(* CODESYS project 车床桁架_RECOVERED_2024-04-08T08-30-31.project
   CompiledLibraryCompatibilityVersion: LeadSysStudio V3.5 SP15 Patch 4
   Title: 车床桁架

Project tree, tasks and I/O mapping:
  Device : SC5-C0A4, Leadshine Technology Co., Ltd., order no. 504001, version 3.5.15.40
    application Application
      libraries: Standard, * (System)
      task MainTask (cyclic, interval t#20ms, priority 1) calls PLC_PRG
      task EtherCAT_Master_Leadshine_A (cyclic, interval 4000 µs, priority 0) calls EtherCAT_Master_Leadshine_A.EtherCAT_Task
      FunctionBlock/
        function block FB102_ClockPuls [LD]
        program Public_Prog [LD]: SystemVar
        function block FB_CylinderDouble [ST]
        function block FB_CylinderSingle [ST]
      global variables HMI_Var
      global variables I_List
      data type CYLINDER_REF
      global variables System
      global variables Publics
      program PLC_PRG [LD]
      global variables O_Lisk
    Device Diagnose
    Network Configuration
      LocalBus Config
    Resource Usage
    LocalBus_Master_Module : LocalBusR1 Master, Leadshine Technology Co., Ltd., version 3.5.15.40
      SC0032N1 : SC0032N1, Leadshine Technology Co., Ltd., version 3.5.15.40
          settings: 位置号 = 1
          unmapped channels: OUTPUT_0, OUTPUT_1, OUTPUT_2, OUTPUT_3
      SC3200 : SC3200, Leadshine Technology Co., Ltd., version 3.5.15.40
          settings: 位置号 = 0
          unmapped channels: INPUT_0, INPUT_1, INPUT_2, INPUT_3
    SoftMotion General Axis Pool
    EtherCAT_Master_Leadshine_A : EtherCAT Master SoftMotion, 3S - Smart Software Solutions GmbH, version 3.5.16.30
        settings: NetworkName = 'ecat'; SelectNetworkByName = TRUE
      L6N_2 : L6N(COE), Leadshine Technology Co.,Ltd., order no. L6N, version Revision=16#00000001
          settings: DC sync0 cycletime = 4000; DC sync1 cycletime = 4000; Number of SDO = 6; Homing method.Index = 16#6098; Homing method.Subindex = 16#00; Homing method.Value = 19; Homing method.Size = 8; Homing method.AbortIfError = FALSE; Homing method.JumpToLine = FALSE; Homing method.Line = 0; Homing method.CompleteAccess = FALSE; Homing velocity (fast).Index = 16#6099; Homing velocity (fast).Subindex = 16#01; Homing velocity (fast).Value = 6103261; Homing velocity (fast).Size = 32; Homing velocity (fast).AbortIfError = FALSE; Homing velocity (fast).JumpToLine = FALSE; Homing velocity (fast).Line = 0; Homing velocity (fast).CompleteAccess = FALSE; Homing velocity (slow).Index = 16#6099; Homing velocity (slow).Subindex = 16#02; Homing velocity (slow).Value = 1220652; Homing velocity (slow).Size = 32; Homing velocity (slow).AbortIfError = FALSE; Homing velocity (slow).JumpToLine = FALSE; Homing velocity (slow).Line = 0; Homing velocity (slow).CompleteAccess = FALSE; Homing acceleration.Index = 16#609A; Homing acceleration.Subindex = 16#00; Homing acceleration.Value = 61032615; Homing acceleration.Size = 32; Homing acceleration.AbortIfError = FALSE; Homing acceleration.JumpToLine = FALSE; Homing acceleration.Line = 0; Homing acceleration.CompleteAccess = FALSE; Homing offset.Index = 16#607C; Homing offset.Subindex = 16#00; Homing offset.Value = 0; Homing offset.Size = 32; Homing offset.AbortIfError = FALSE;
            Homing offset.JumpToLine = FALSE; Homing offset.Line = 0; Homing offset.CompleteAccess = FALSE
          unmapped channels: Control word, Profile target position, Touch Probe Function, Last error code, Status word, Modes of operation display, Position loop error, Actual motor torque, Actual motor position, Touch Probe Status, Touch probe pos1 pos value, Digital inputs
        Axis_2 : Axis, 3S - Smart Software Solutions GmbH, order no. 0, version 4.6.1.0
            settings: wDriveID = 2; dwRatioTechUnitsDenom = 610326149; iRatioTechUnitsNum = 1000; fSWMaxVelocity = 1000; fSWMaxAcceleration = 10000; fSWMaxDeceleration = 10000; fSWMaxJerk = 100000; 一圈脉冲数 = 8388608; 工作台一圈的位移 = 109.955741; 电子齿轮比分子 = 8; 电子齿轮比分母 = 1; ScalingIncs = 8388608; ScalingMotorTurns2 = 8; AdrOffset_8010 = 28; BitOffset_8010 = 0; BitLength_8010 = 16; Address_8010 = '%QW14'; Type_8010 = 'UINT'; AddressPointer_8010 = ADR(%QW14); AdrOffset_8020 = 32; BitOffset_8020 = 0; BitLength_8020 = 32; Address_8020 = '%QD8'; Type_8020 = 'DINT'; AddressPointer_8020 = ADR(%QD8); AdrOffset_8030 = 4294967295; BitOffset_8030 = 0; BitLength_8030 = 32; Address_8030 = ''; Type_8030 = 'DINT'; AddressPointer_8030 = 0; AdrOffset_8040 = 4294967295; BitOffset_8040 = 0; BitLength_8040 = 16; Address_8040 = ''; Type_8040 = 'INT'; AddressPointer_8040 = 0; AdrOffset_8050 = 4294967295; BitOffset_8050 = 0; BitLength_8050 = 8;
              Address_8050 = ''; Type_8050 = 'SINT'; AddressPointer_8050 = 0; AdrOffset_8060 = 36; BitOffset_8060 = 0; BitLength_8060 = 16; Address_8060 = '%QW18'; Type_8060 = 'UINT'; AddressPointer_8060 = ADR(%QW18); AdrOffset_8070 = 4294967295; BitOffset_8070 = 0; BitLength_8070 = 0; Address_8070 = ''; Type_8070 = ''; AddressPointer_8070 = 0; AdrOffset_8080 = 4294967295; BitOffset_8080 = 0; BitLength_8080 = 16; Address_8080 = ''; Type_8080 = 'INT'; AddressPointer_8080 = 0; AdrOffset_8090 = 4294967295; BitOffset_8090 = 0; BitLength_8090 = 0; Address_8090 = ''; Type_8090 = ''; AddressPointer_8090 = 0; AdrOffset_8510 = 70; BitOffset_8510 = 0; BitLength_8510 = 16; Address_8510 = '%IW35'; Type_8510 = 'UINT'; AddressPointer_8510 = ADR(%IW35); AdrOffset_8520 = 84; BitOffset_8520 = 0; BitLength_8520 = 32; Address_8520 = '%ID21'; Type_8520 = 'DINT'; AddressPointer_8520 = ADR(%ID21); AdrOffset_8530 = 4294967295;
              BitOffset_8530 = 0; BitLength_8530 = 0; Address_8530 = ''; Type_8530 = ''; AddressPointer_8530 = 0; AdrOffset_8540 = 80; BitOffset_8540 = 0; BitLength_8540 = 16; Address_8540 = '%IW40'; Type_8540 = 'INT'; AddressPointer_8540 = ADR(%IW40); AdrOffset_8550 = 72; BitOffset_8550 = 0; BitLength_8550 = 8; Address_8550 = '%IB72'; Type_8550 = 'SINT'; AddressPointer_8550 = ADR(%IB72); AdrOffset_8560 = 96; BitOffset_8560 = 0; BitLength_8560 = 32; Address_8560 = '%ID24'; Type_8560 = 'UDINT'; AddressPointer_8560 = ADR(%ID24); AdrOffset_8570 = 88; BitOffset_8570 = 0; BitLength_8570 = 16; Address_8570 = '%IW44'; Type_8570 = 'UINT'; AddressPointer_8570 = ADR(%IW44); AdrOffset_8580 = 92; BitOffset_8580 = 0; BitLength_8580 = 32; Address_8580 = '%ID23'; Type_8580 = 'DINT'; AddressPointer_8580 = ADR(%ID23); AdrOffset_8590 = 4294967295; BitOffset_8590 = 0; BitLength_8590 = 0; Address_8590 = ''; Type_8590 = '';
              AddressPointer_8590 = 0; AdrOffset_8600 = 4294967295; BitOffset_8600 = 0; BitLength_8600 = 0; Address_8600 = ''; Type_8600 = ''; AddressPointer_8600 = 0; AdrOffset_8600 = 4294967295; BitOffset_8600 = 0; BitLength_8600 = 0; Address_8610 = ''; Type_8610 = ''; AddressPointer_8610 = 0; AdrOffset_8620 = 76; BitOffset_8620 = 0; BitLength_8620 = 32; Address_8620 = '%ID19'; Type_8620 = 'DINT'; AddressPointer_8620 = ADR(%ID19)
      L6N_3 : L6N(COE), Leadshine Technology Co.,Ltd., order no. L6N, version Revision=16#00000001
          settings: DC sync0 cycletime = 4000; DC sync1 cycletime = 4000; Number of SDO = 6; Homing method.Index = 16#6098; Homing method.Subindex = 16#00; Homing method.Value = 19; Homing method.Size = 8; Homing method.AbortIfError = FALSE; Homing method.JumpToLine = FALSE; Homing method.Line = 0; Homing method.CompleteAccess = FALSE; Homing velocity (fast).Index = 16#6099; Homing velocity (fast).Subindex = 16#01; Homing velocity (fast).Value = 26701769; Homing velocity (fast).Size = 32; Homing velocity (fast).AbortIfError = FALSE; Homing velocity (fast).JumpToLine = FALSE; Homing velocity (fast).Line = 0; Homing velocity (fast).CompleteAccess = FALSE; Homing velocity (slow).Index = 16#6099; Homing velocity (slow).Subindex = 16#02; Homing velocity (slow).Value = 5340354; Homing velocity (slow).Size = 32; Homing velocity (slow).AbortIfError = FALSE; Homing velocity (slow).JumpToLine = FALSE; Homing velocity (slow).Line = 0; Homing velocity (slow).CompleteAccess = FALSE; Homing acceleration.Index = 16#609A; Homing acceleration.Subindex = 16#00; Homing acceleration.Value = 267017690; Homing acceleration.Size = 32; Homing acceleration.AbortIfError = FALSE; Homing acceleration.JumpToLine = FALSE; Homing acceleration.Line = 0; Homing acceleration.CompleteAccess = FALSE; Homing offset.Index = 16#607C; Homing offset.Subindex = 16#00; Homing offset.Value = 0; Homing offset.Size = 32; Homing offset.AbortIfError = FALSE;
            Homing offset.JumpToLine = FALSE; Homing offset.Line = 0; Homing offset.CompleteAccess = FALSE
          unmapped channels: Control word, Profile target position, Touch Probe Function, Last error code, Status word, Modes of operation display, Position loop error, Actual motor torque, Actual motor position, Touch Probe Status, Touch probe pos1 pos value, Digital inputs
        Axis_3 : Axis, 3S - Smart Software Solutions GmbH, order no. 0, version 4.6.1.0
            settings: wDriveID = 3; dwRatioTechUnitsDenom = 26701769; iRatioTechUnitsNum = 10; fSWMaxVelocity = 1000; fSWMaxAcceleration = 10000; fSWMaxDeceleration = 10000; fSWMaxJerk = 100000; 一圈脉冲数 = 8388608; 工作台一圈的位移 = 109.955741; 电子齿轮比分子 = 35; 电子齿轮比分母 = 1; ScalingIncs = 8388608; ScalingMotorTurns2 = 35; AdrOffset_8010 = 40; BitOffset_8010 = 0; BitLength_8010 = 16; Address_8010 = '%QW20'; Type_8010 = 'UINT'; AddressPointer_8010 = ADR(%QW20); AdrOffset_8020 = 44; BitOffset_8020 = 0; BitLength_8020 = 32; Address_8020 = '%QD11'; Type_8020 = 'DINT'; AddressPointer_8020 = ADR(%QD11); AdrOffset_8030 = 4294967295; BitOffset_8030 = 0; BitLength_8030 = 32; Address_8030 = ''; Type_8030 = 'DINT'; AddressPointer_8030 = 0; AdrOffset_8040 = 4294967295; BitOffset_8040 = 0; BitLength_8040 = 16; Address_8040 = ''; Type_8040 = 'INT'; AddressPointer_8040 = 0; AdrOffset_8050 = 4294967295; BitOffset_8050 = 0; BitLength_8050 = 8;
              Address_8050 = ''; Type_8050 = 'SINT'; AddressPointer_8050 = 0; AdrOffset_8060 = 48; BitOffset_8060 = 0; BitLength_8060 = 16; Address_8060 = '%QW24'; Type_8060 = 'UINT'; AddressPointer_8060 = ADR(%QW24); AdrOffset_8070 = 4294967295; BitOffset_8070 = 0; BitLength_8070 = 0; Address_8070 = ''; Type_8070 = ''; AddressPointer_8070 = 0; AdrOffset_8080 = 4294967295; BitOffset_8080 = 0; BitLength_8080 = 16; Address_8080 = ''; Type_8080 = 'INT'; AddressPointer_8080 = 0; AdrOffset_8090 = 4294967295; BitOffset_8090 = 0; BitLength_8090 = 0; Address_8090 = ''; Type_8090 = ''; AddressPointer_8090 = 0; AdrOffset_8510 = 102; BitOffset_8510 = 0; BitLength_8510 = 16; Address_8510 = '%IW51'; Type_8510 = 'UINT'; AddressPointer_8510 = ADR(%IW51); AdrOffset_8520 = 116; BitOffset_8520 = 0; BitLength_8520 = 32; Address_8520 = '%ID29'; Type_8520 = 'DINT'; AddressPointer_8520 = ADR(%ID29); AdrOffset_8530 = 4294967295;
              BitOffset_8530 = 0; BitLength_8530 = 0; Address_8530 = ''; Type_8530 = ''; AddressPointer_8530 = 0; AdrOffset_8540 = 112; BitOffset_8540 = 0; BitLength_8540 = 16; Address_8540 = '%IW56'; Type_8540 = 'INT'; AddressPointer_8540 = ADR(%IW56); AdrOffset_8550 = 104; BitOffset_8550 = 0; BitLength_8550 = 8; Address_8550 = '%IB104'; Type_8550 = 'SINT'; AddressPointer_8550 = ADR(%IB104); AdrOffset_8560 = 128; BitOffset_8560 = 0; BitLength_8560 = 32; Address_8560 = '%ID32'; Type_8560 = 'UDINT'; AddressPointer_8560 = ADR(%ID32); AdrOffset_8570 = 120; BitOffset_8570 = 0; BitLength_8570 = 16; Address_8570 = '%IW60'; Type_8570 = 'UINT'; AddressPointer_8570 = ADR(%IW60); AdrOffset_8580 = 124; BitOffset_8580 = 0; BitLength_8580 = 32; Address_8580 = '%ID31'; Type_8580 = 'DINT'; AddressPointer_8580 = ADR(%ID31); AdrOffset_8590 = 4294967295; BitOffset_8590 = 0; BitLength_8590 = 0; Address_8590 = ''; Type_8590 = '';
              AddressPointer_8590 = 0; AdrOffset_8600 = 4294967295; BitOffset_8600 = 0; BitLength_8600 = 0; Address_8600 = ''; Type_8600 = ''; AddressPointer_8600 = 0; AdrOffset_8600 = 4294967295; BitOffset_8600 = 0; BitLength_8600 = 0; Address_8610 = ''; Type_8610 = ''; AddressPointer_8610 = 0; AdrOffset_8620 = 108; BitOffset_8620 = 0; BitLength_8620 = 32; Address_8620 = '%ID27'; Type_8620 = 'DINT'; AddressPointer_8620 = ADR(%ID27)
      L6N_1 : L6N(COE), Leadshine Technology Co.,Ltd., order no. L6N, version Revision=16#00000001
          settings: DC sync0 cycletime = 4000; DC sync1 cycletime = 4000; Number of SDO = 6; Homing method.Index = 16#6098; Homing method.Subindex = 16#00; Homing method.Value = 19; Homing method.Size = 8; Homing method.AbortIfError = FALSE; Homing method.JumpToLine = FALSE; Homing method.Line = 0; Homing method.CompleteAccess = FALSE; Homing velocity (fast).Index = 16#6099; Homing velocity (fast).Subindex = 16#01; Homing velocity (fast).Value = 16777216; Homing velocity (fast).Size = 32; Homing velocity (fast).AbortIfError = FALSE; Homing velocity (fast).JumpToLine = FALSE; Homing velocity (fast).Line = 0; Homing velocity (fast).CompleteAccess = FALSE; Homing velocity (slow).Index = 16#6099; Homing velocity (slow).Subindex = 16#02; Homing velocity (slow).Value = 3355443; Homing velocity (slow).Size = 32; Homing velocity (slow).AbortIfError = FALSE; Homing velocity (slow).JumpToLine = FALSE; Homing velocity (slow).Line = 0; Homing velocity (slow).CompleteAccess = FALSE; Homing acceleration.Index = 16#609A; Homing acceleration.Subindex = 16#00; Homing acceleration.Value = 167772160; Homing acceleration.Size = 32; Homing acceleration.AbortIfError = FALSE; Homing acceleration.JumpToLine = FALSE; Homing acceleration.Line = 0; Homing acceleration.CompleteAccess = FALSE; Homing offset.Index = 16#607C; Homing offset.Subindex = 16#00; Homing offset.Value = 0; Homing offset.Size = 32; Homing offset.AbortIfError = FALSE;
            Homing offset.JumpToLine = FALSE; Homing offset.Line = 0; Homing offset.CompleteAccess = FALSE
          unmapped channels: Control word, Profile target position, Touch Probe Function, Last error code, Status word, Modes of operation display, Position loop error, Actual motor torque, Actual motor position, Touch Probe Status, Touch probe pos1 pos value, Digital inputs
        Axis_1 : Axis, 3S - Smart Software Solutions GmbH, order no. 0, version 4.6.1.0
            settings: dwRatioTechUnitsDenom = 8388608; iRatioTechUnitsNum = 5; fSWMaxVelocity = 1000; fSWMaxAcceleration = 10000; fSWMaxDeceleration = 10000; fSWMaxJerk = 100000; 一圈脉冲数 = 8388608; 工作台一圈的位移 = 5; 电子齿轮比分子 = 1; 电子齿轮比分母 = 1; ScalingIncs = 8388608; AdrOffset_8010 = 16; BitOffset_8010 = 0; BitLength_8010 = 16; Address_8010 = '%QW8'; Type_8010 = 'UINT'; AddressPointer_8010 = ADR(%QW8); AdrOffset_8020 = 20; BitOffset_8020 = 0; BitLength_8020 = 32; Address_8020 = '%QD5'; Type_8020 = 'DINT'; AddressPointer_8020 = ADR(%QD5); AdrOffset_8030 = 4294967295; BitOffset_8030 = 0; BitLength_8030 = 32; Address_8030 = ''; Type_8030 = 'DINT'; AddressPointer_8030 = 0; AdrOffset_8040 = 4294967295; BitOffset_8040 = 0; BitLength_8040 = 16; Address_8040 = ''; Type_8040 = 'INT'; AddressPointer_8040 = 0; AdrOffset_8050 = 4294967295; BitOffset_8050 = 0; BitLength_8050 = 8; Address_8050 = ''; Type_8050 = 'SINT';
              AddressPointer_8050 = 0; AdrOffset_8060 = 24; BitOffset_8060 = 0; BitLength_8060 = 16; Address_8060 = '%QW12'; Type_8060 = 'UINT'; AddressPointer_8060 = ADR(%QW12); AdrOffset_8070 = 4294967295; BitOffset_8070 = 0; BitLength_8070 = 0; Address_8070 = ''; Type_8070 = ''; AddressPointer_8070 = 0; AdrOffset_8080 = 4294967295; BitOffset_8080 = 0; BitLength_8080 = 16; Address_8080 = ''; Type_8080 = 'INT'; AddressPointer_8080 = 0; AdrOffset_8090 = 4294967295; BitOffset_8090 = 0; BitLength_8090 = 0; Address_8090 = ''; Type_8090 = ''; AddressPointer_8090 = 0; AdrOffset_8510 = 38; BitOffset_8510 = 0; BitLength_8510 = 16; Address_8510 = '%IW19'; Type_8510 = 'UINT'; AddressPointer_8510 = ADR(%IW19); AdrOffset_8520 = 52; BitOffset_8520 = 0; BitLength_8520 = 32; Address_8520 = '%ID13'; Type_8520 = 'DINT'; AddressPointer_8520 = ADR(%ID13); AdrOffset_8530 = 4294967295; BitOffset_8530 = 0; BitLength_8530 = 0;
              Address_8530 = ''; Type_8530 = ''; AddressPointer_8530 = 0; AdrOffset_8540 = 48; BitOffset_8540 = 0; BitLength_8540 = 16; Address_8540 = '%IW24'; Type_8540 = 'INT'; AddressPointer_8540 = ADR(%IW24); AdrOffset_8550 = 40; BitOffset_8550 = 0; BitLength_8550 = 8; Address_8550 = '%IB40'; Type_8550 = 'SINT'; AddressPointer_8550 = ADR(%IB40); AdrOffset_8560 = 64; BitOffset_8560 = 0; BitLength_8560 = 32; Address_8560 = '%ID16'; Type_8560 = 'UDINT'; AddressPointer_8560 = ADR(%ID16); AdrOffset_8570 = 56; BitOffset_8570 = 0; BitLength_8570 = 16; Address_8570 = '%IW28'; Type_8570 = 'UINT'; AddressPointer_8570 = ADR(%IW28); AdrOffset_8580 = 60; BitOffset_8580 = 0; BitLength_8580 = 32; Address_8580 = '%ID15'; Type_8580 = 'DINT'; AddressPointer_8580 = ADR(%ID15); AdrOffset_8590 = 4294967295; BitOffset_8590 = 0; BitLength_8590 = 0; Address_8590 = ''; Type_8590 = ''; AddressPointer_8590 = 0; AdrOffset_8600 = 4294967295;
              BitOffset_8600 = 0; BitLength_8600 = 0; Address_8600 = ''; Type_8600 = ''; AddressPointer_8600 = 0; AdrOffset_8600 = 4294967295; BitOffset_8600 = 0; BitLength_8600 = 0; Address_8610 = ''; Type_8610 = ''; AddressPointer_8610 = 0; AdrOffset_8620 = 44; BitOffset_8620 = 0; BitLength_8620 = 32; Address_8620 = '%ID11'; Type_8620 = 'DINT'; AddressPointer_8620 = ADR(%ID11)
      L6N : L6N(COE), Leadshine Technology Co.,Ltd., order no. L6N, version Revision=16#00000001
          settings: DC sync0 cycletime = 4000; DC enable = 1; DC sync0 enable = 1; DC sync0 shift time = 0; DC sync1 cycletime = 4000; DC sync1 enable = 0; DC sync1 factor = 'x 1'; DC sync1 shift time = 0; Number of SDO = 6; Homing method.Index = 16#6098; Homing method.Subindex = 16#00; Homing method.Value = 30; Homing method.Size = 8; Homing method.AbortIfError = FALSE; Homing method.JumpToLine = FALSE; Homing method.Line = 0; Homing method.CompleteAccess = FALSE; Homing velocity (fast).Index = 16#6099; Homing velocity (fast).Subindex = 16#01; Homing velocity (fast).Value = 20971520; Homing velocity (fast).Size = 32; Homing velocity (fast).AbortIfError = FALSE; Homing velocity (fast).JumpToLine = FALSE; Homing velocity (fast).Line = 0; Homing velocity (fast).CompleteAccess = FALSE; Homing velocity (slow).Index = 16#6099; Homing velocity (slow).Subindex = 16#02; Homing velocity (slow).Value = 4194304; Homing velocity (slow).Size = 32; Homing velocity (slow).AbortIfError = FALSE; Homing velocity (slow).JumpToLine = FALSE; Homing velocity (slow).Line = 0; Homing velocity (slow).CompleteAccess = FALSE; Homing acceleration.Index = 16#609A; Homing acceleration.Subindex = 16#00; Homing acceleration.Value = 209715200; Homing acceleration.Size = 32; Homing acceleration.AbortIfError = FALSE; Homing acceleration.JumpToLine = FALSE; Homing acceleration.Line = 0;
            Homing acceleration.CompleteAccess = FALSE; Homing offset.Index = 16#607C; Homing offset.Subindex = 16#00; Homing offset.Value = 0; Homing offset.Size = 32; Homing offset.AbortIfError = FALSE; Homing offset.JumpToLine = FALSE; Homing offset.Line = 0; Homing offset.CompleteAccess = FALSE
          unmapped channels: Control word, Profile target position, Touch Probe Function, Last error code, Status word, Modes of operation display, Position loop error, Actual motor torque, Actual motor position, Touch Probe Status, Touch probe pos1 pos value, Digital inputs
        Axis : Axis, 3S - Smart Software Solutions GmbH, order no. 0, version 4.6.1.0
            settings: wDriveID = 0; dwRatioTechUnitsDenom = 2097152; fSWMaxVelocity = 1000; fSWMaxAcceleration = 10000; fSWMaxDeceleration = 10000; fSWMaxJerk = 100000; 一圈脉冲数 = 8388608; 工作台一圈的位移 = 4; 电子齿轮比分子 = 1; 电子齿轮比分母 = 1; ScalingIncs = 8388608; AdrOffset_8010 = 4; BitOffset_8010 = 0; BitLength_8010 = 16; Address_8010 = '%QW2'; Type_8010 = 'UINT'; AddressPointer_8010 = ADR(%QW2); AdrOffset_8020 = 8; BitOffset_8020 = 0; BitLength_8020 = 32; Address_8020 = '%QD2'; Type_8020 = 'DINT'; AddressPointer_8020 = ADR(%QD2); AdrOffset_8030 = 4294967295; BitOffset_8030 = 0; BitLength_8030 = 32; Address_8030 = ''; Type_8030 = 'DINT'; AddressPointer_8030 = 0; AdrOffset_8040 = 4294967295; BitOffset_8040 = 0; BitLength_8040 = 16; Address_8040 = ''; Type_8040 = 'INT'; AddressPointer_8040 = 0; AdrOffset_8050 = 4294967295; BitOffset_8050 = 0; BitLength_8050 = 8; Address_8050 = ''; Type_8050 = 'SINT';
              AddressPointer_8050 = 0; AdrOffset_8060 = 12; BitOffset_8060 = 0; BitLength_8060 = 16; Address_8060 = '%QW6'; Type_8060 = 'UINT'; AddressPointer_8060 = ADR(%QW6); AdrOffset_8070 = 4294967295; BitOffset_8070 = 0; BitLength_8070 = 0; Address_8070 = ''; Type_8070 = ''; AddressPointer_8070 = 0; AdrOffset_8080 = 4294967295; BitOffset_8080 = 0; BitLength_8080 = 16; Address_8080 = ''; Type_8080 = 'INT'; AddressPointer_8080 = 0; AdrOffset_8090 = 4294967295; BitOffset_8090 = 0; BitLength_8090 = 0; Address_8090 = ''; Type_8090 = ''; AddressPointer_8090 = 0; AdrOffset_8510 = 6; BitOffset_8510 = 0; BitLength_8510 = 16; Address_8510 = '%IW3'; Type_8510 = 'UINT'; AddressPointer_8510 = ADR(%IW3); AdrOffset_8520 = 20; BitOffset_8520 = 0; BitLength_8520 = 32; Address_8520 = '%ID5'; Type_8520 = 'DINT'; AddressPointer_8520 = ADR(%ID5); AdrOffset_8530 = 4294967295; BitOffset_8530 = 0; BitLength_8530 = 0;
              Address_8530 = ''; Type_8530 = ''; AddressPointer_8530 = 0; AdrOffset_8540 = 16; BitOffset_8540 = 0; BitLength_8540 = 16; Address_8540 = '%IW8'; Type_8540 = 'INT'; AddressPointer_8540 = ADR(%IW8); AdrOffset_8550 = 8; BitOffset_8550 = 0; BitLength_8550 = 8; Address_8550 = '%IB8'; Type_8550 = 'SINT'; AddressPointer_8550 = ADR(%IB8); AdrOffset_8560 = 32; BitOffset_8560 = 0; BitLength_8560 = 32; Address_8560 = '%ID8'; Type_8560 = 'UDINT'; AddressPointer_8560 = ADR(%ID8); AdrOffset_8570 = 24; BitOffset_8570 = 0; BitLength_8570 = 16; Address_8570 = '%IW12'; Type_8570 = 'UINT'; AddressPointer_8570 = ADR(%IW12); AdrOffset_8580 = 28; BitOffset_8580 = 0; BitLength_8580 = 32; Address_8580 = '%ID7'; Type_8580 = 'DINT'; AddressPointer_8580 = ADR(%ID7); AdrOffset_8590 = 4294967295; BitOffset_8590 = 0; BitLength_8590 = 0; Address_8590 = ''; Type_8590 = ''; AddressPointer_8590 = 0; AdrOffset_8600 = 4294967295;
              BitOffset_8600 = 0; BitLength_8600 = 0; Address_8600 = ''; Type_8600 = ''; AddressPointer_8600 = 0; AdrOffset_8600 = 4294967295; BitOffset_8600 = 0; BitLength_8600 = 0; Address_8610 = ''; Type_8610 = ''; AddressPointer_8610 = 0; AdrOffset_8620 = 12; BitOffset_8620 = 0; BitLength_8620 = 32; Address_8620 = '%ID3'; Type_8620 = 'DINT'; AddressPointer_8620 = ADR(%ID3)
*)

// Device/Application/CYLINDER_REF
TYPE CYLINDER_REF :
STRUCT
	///初始化时返回原位控制
	xInit: BOOL;
	///自动控制,变为TRUE时，执行到位控制，变为FALSE时执行原位控制
	xAutoCmd: BOOL;
	///到位标志,处于原位状态
	xIsBack: BOOL;
	///到位标志,处于到位状态	
	xIsFront: BOOL;
END_STRUCT
END_TYPE

// Device/Application/HMI_Var
{attribute 'qualified_only'}
VAR_GLOBAL
END_VAR

// Device/Application/I_List
{attribute 'qualified_only'}
VAR_GLOBAL
	// 上料传送带到位确认
	X0 AT %IX0.0: BOOL;
	// 紧急停止
	X1 AT %IX0.1: BOOL;
	// 推出气缸原位
	X2 AT %IX0.2: BOOL;
	// 推出气缸动作位
	X3 AT %IX0.3: BOOL;
	// 顶起气缸原位
	X4 AT %IX0.4: BOOL;
	// 顶起气缸动作位
	X5 AT %IX0.5: BOOL;
	// 上料气爪原位
	X6 AT %IX0.6: BOOL;
	// 上料气爪动作位
	X7 AT %IX0.7: BOOL;
	// 下料气爪原位
	X10 AT %IX1.0: BOOL;
	// 下料气爪动作位
	X11 AT %IX1.1: BOOL;
	// 翻转气缸原位
	X12 AT %IX1.2: BOOL;
	// 翻转气缸动作位
	X13 AT %IX1.3: BOOL;
	// 开门气缸原位
	X14 AT %IX1.4: BOOL;
	// 开门气缸动作位
	X15 AT %IX1.5: BOOL;
	// 启动按钮
	X16 AT %IX1.6: BOOL;
	// 停止按钮
	X17 AT %IX1.7: BOOL;
	// 复位按钮
	X20 AT %IX2.0: BOOL;
	// 手自动按钮ON为自动
	X21 AT %IX2.1: BOOL;
	// 下料确认
	X22 AT %IX2.2: BOOL;
	// 联机卡盘夹紧
	X23 AT %IX2.3: BOOL;
	// 联机启动
	X24 AT %IX2.4: BOOL;
	// 联机停止
	X25 AT %IX2.5: BOOL;
	// 联机故障
	X26 AT %IX2.6: BOOL;
	// 联机X轴零点
	X27 AT %IX2.7: BOOL;
	// 联机Z轴零点
	X30 AT %IX3.0: BOOL;
	X31 AT %IX3.1: BOOL;
	X32 AT %IX3.2: BOOL;
	X33 AT %IX3.3: BOOL;
	X34 AT %IX3.4: BOOL;
	X35 AT %IX3.5: BOOL;
	X36 AT %IX3.6: BOOL;
	X37 AT %IX3.7: BOOL;
END_VAR

// Device/Application/System
{attribute 'qualified_only'}
VAR_GLOBAL
	// 上电扫描一周期
FirstScan    :BOOL;
// 常ON
AlwaysTRUE   : BOOL;
// 常OFF
AlwaysFALSE  : BOOL;
// 0.1S周期脉冲
Clock_10Hz    :BOOL;
// 0.2S周期脉冲
Clock_5Hz    :BOOL;
// 0.5S周期脉冲
Clock_2Hz    :BOOL;
// 1S周期脉冲
Clock_1Hz    :BOOL;
// 2S周期脉冲
Clock_HalfHz :BOOL;
END_VAR

// Device/Application/Publics
{attribute 'qualified_only'}
VAR_GLOBAL
	// 调试使用常ON
CYGIA_ON   :BOOL;
// 调试使用常OFF
CYGIA_OFF  :BOOL;
END_VAR

// Device/Application/O_Lisk
{attribute 'qualified_only'}
VAR_GLOBAL
	// 皮带运转
	Y0 AT %QX0.0: BOOL;
	// 震动筛运动
	Y1 AT %QX0.1: BOOL;
	// 推出气缸原位
	Y2 AT %QX0.2: BOOL;
	// 紧急停止输出
	Y3 AT %QX0.3: BOOL;
	// 顶起气缸原位
	Y4 AT %QX0.4: BOOL;
	Y5 AT %QX0.5: BOOL;
	// 上料气爪原位
	Y6 AT %QX0.6: BOOL;
	Y7 AT %QX0.7: BOOL;
	// 下料气爪原位
	Y10 AT %QX1.0: BOOL;
	Y11 AT %QX1.0: BOOL;
	// 翻转气缸原位
	Y12 AT %QX1.0: BOOL;
	Y13 AT %QX1.0: BOOL;
	// 开门气缸原位
	Y14 AT %QX1.0: BOOL;
	Y15 AT %QX1.5: BOOL;
	// 启动按钮LED
	Y16 AT %QX1.6: BOOL;
	// 停止按钮LED
	Y17 AT %QX1.7: BOOL;
	// 复位按钮LED
	Y20 AT %QX2.0: BOOL;
	Y21 AT %QX2.1: BOOL;
	// 下料传送带
	Y22 AT %QX2.2: BOOL;
	// 三色灯红
	Y23 AT %QX2.3: BOOL;
	// 三色灯黄
	Y24 AT %QX2.4: BOOL;
	// 三色灯绿
	Y25 AT %QX2.5: BOOL;
	// 三色灯蜂鸣
	Y26 AT %QX2.6: BOOL;
	// 联机卡盘夹紧
	Y27 AT %QX2.7: BOOL;
	// 联机启动
	Y30 AT %QX3.0: BOOL;
	// 联机停止
	Y31 AT %QX3.1: BOOL;
	Y32 AT %QX3.2: BOOL;
	Y33 AT %QX3.3: BOOL;
	Y34 AT %QX3.4: BOOL;
	Y35 AT %QX3.5: BOOL;
	Y36 AT %QX3.6: BOOL;
	Y37 AT %QX3.7: BOOL;
END_VAR

// Device/Application/PLC_PRG
PROGRAM PLC_PRG
VAR
	SMC3_ReinitDrive_0: SMC3_ReinitDrive;
END_VAR

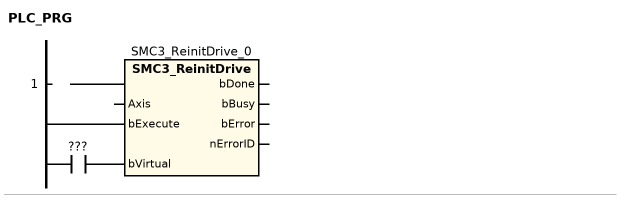
// NETWORK 1
SMC3_ReinitDrive_0(bExecute := TRUE); // SMC3_ReinitDrive

END_PROGRAM

// Device/Application/FunctionBlock/FB102_ClockPuls
FUNCTION_BLOCK FB102_ClockPuls
VAR_INPUT
	///脉冲ON时间
	iTimeON: TIME;
	///脉冲OFF时间
	iTimeOFF: TIME;
END_VAR
VAR_OUTPUT
	///时钟脉冲差速器
	oClockVar: BOOL;
END_VAR
VAR
	TON_Clock: TON;
	TOF_Clock: TOF;
END_VAR

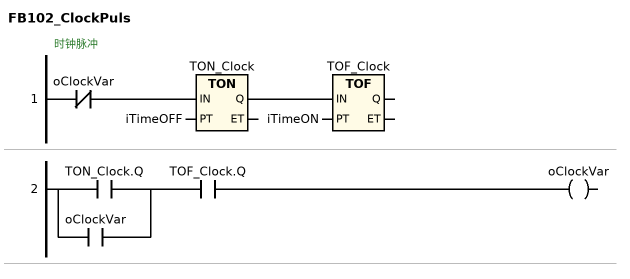
// NETWORK 1
// 时钟脉冲
TON_Clock(IN := NOT oClockVar, PT := iTimeOFF); // TON
TOF_Clock(IN := TON_Clock.Q, PT := iTimeON); // TOF

// NETWORK 2
oClockVar := (TON_Clock.Q OR oClockVar) AND TOF_Clock.Q;

END_FUNCTION_BLOCK

// Device/Application/FunctionBlock/Public_Prog
PROGRAM Public_Prog
VAR
	Clock_10Hz: FB102_ClockPuls;
	Clock_5Hz: FB102_ClockPuls;
	Clock_2Hz: FB102_ClockPuls;
	Clock_1Hz: FB102_ClockPuls;
	Clock_HalfHz: FB102_ClockPuls;
END_VAR
VAR // added by the converter: edge detectors and wires of the graphical bodies
    _rt1 : R_TRIG;
END_VAR

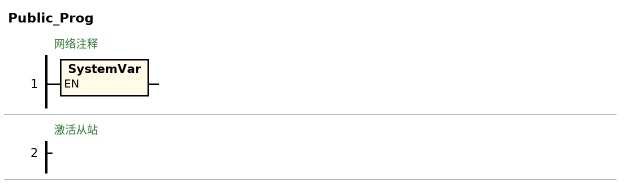
// NETWORK 1
// 网络注释
SystemVar();

// NETWORK 2
// 激活从站

ACTION SystemVar:
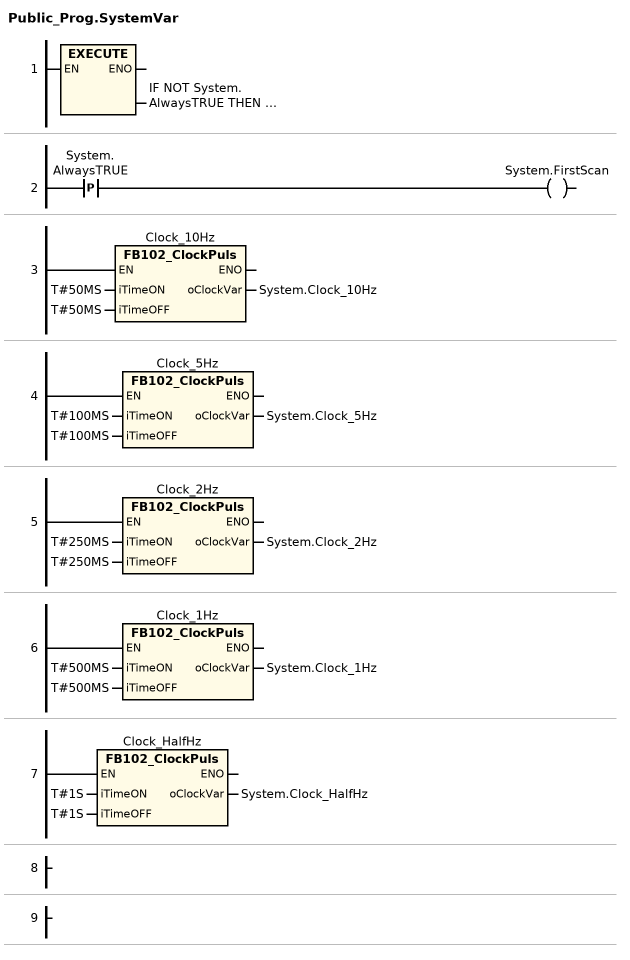
// NETWORK 1
IF NOT System.AlwaysTRUE THEN
	System.AlwaysTRUE := TRUE;
END_IF
IF  System.AlwaysFALSE THEN
	System.AlwaysFALSE := FALSE;
END_IF
IF NOT Publics.CYGIA_ON THEN
	Publics.CYGIA_ON := TRUE;
END_IF
IF  Publics.CYGIA_OFF THEN
	Publics.CYGIA_OFF := FALSE;
END_IF

// NETWORK 2
_rt1(CLK := System.AlwaysTRUE);
System.FirstScan := _rt1.Q;

// NETWORK 3
Clock_10Hz(iTimeON := T#50MS, iTimeOFF := T#50MS, oClockVar => System.Clock_10Hz); // FB102_ClockPuls

// NETWORK 4
Clock_5Hz(iTimeON := T#100MS, iTimeOFF := T#100MS, oClockVar => System.Clock_5Hz); // FB102_ClockPuls

// NETWORK 5
Clock_2Hz(iTimeON := T#250MS, iTimeOFF := T#250MS, oClockVar => System.Clock_2Hz); // FB102_ClockPuls

// NETWORK 6
Clock_1Hz(iTimeON := T#500MS, iTimeOFF := T#500MS, oClockVar => System.Clock_1Hz); // FB102_ClockPuls

// NETWORK 7
Clock_HalfHz(iTimeON := T#1S, iTimeOFF := T#1S, oClockVar => System.Clock_HalfHz); // FB102_ClockPuls

// NETWORK 8

// NETWORK 9
END_ACTION

END_PROGRAM

// Device/Application/FunctionBlock/FB_CylinderDouble
FUNCTION_BLOCK FB_CylinderDouble
VAR_IN_OUT
	///气缸控制、状态和报警
	stCylvar: CYLINDER_REF;
END_VAR
VAR_INPUT
	///安全条件
	xReady: BOOL;
	///报警复位
	xReset: BOOL;
	///手动控制,每on一次,则反转输出点状态
	xManuCmd: BOOL;
	///原位检测
	xBackSensor: BOOL;
	///到位检测
	xFrontSensor: BOOL;
	///手自动不一致报警无效
	xManuAlmDisable: BOOL;
	///原位检测无效
	xBackSensorDisable: BOOL;
	///到位检测无效	
	xFrontSensorDisable: BOOL;
	///原位延时	
	wBackDelay: WORD;
	///到位延时
	wFrontDelay: WORD;
END_VAR
VAR_OUTPUT
	///输出点,对应双控气缸原位电磁阀
	xOutputA: BOOL;
	///输出点,应双控气缸到位电磁阀
	xOutputB: BOOL;
	///未满足安全条件报警
	f_xNotRdyAlm: BOOL;
	///手自动不一致报警	
	f_xManuAlm: BOOL;
	///未在原位报警
	f_xBackAlm: BOOL;
	///未到位报警	
	f_xFrontAlm: BOOL;
	///气缸处于不受控制状态报警
	f_xUncontrolledAlm: BOOL;
END_VAR
VAR
	///获取自动控制的上升沿
	fbAutoRise: R_TRIG;
	///获取自动控制的下升沿
	fbAutoFall: F_TRIG;
	///获取手动控制的下升沿
	fbManuFall: F_TRIG;
	///获取复位信号的上升沿
	fbResetRise: R_TRIG;
	///原位状态延时,用于输出原位状态
	fbBackTon: TON;
	///到位状态延时,用于输出到位状态	
	fbFrontTon: TON;
	///获取原位状态下降沿
	fbBackFall: F_TRIG;
	///获取到位状态下降沿
	fbFrontFall: F_TRIG;
	///原位动作超时,用于输出未在原位位置报警
	fbBackWait: TON;
	///到位动作超时,用于输出未在原位位置报警
	fbFrontWait: TON;
END_VAR

   //初始化时返回原位
   IF  xReady AND stCylvar.xInit AND ( NOT xManuCmd ) THEN
	     xOutputA  := TRUE; 
         xOutputB  := FALSE;
		 f_xManuAlm  := FALSE;
		 stCylvar.xInit  := FALSE;	  	  	 	  
   END_IF	  
   
   //获取手动控制、自动控制的边沿信号
   fbManuFall(CLK:=xManuCmd , Q=> );
   fbAutoRise(CLK:=stCylvar.xAutoCmd , Q=> );
   fbAutoFall(CLK:=stCylvar.xAutoCmd , Q=> );
   
   //1,手动操作时，如果满足安全条件且未屏蔽手自动不一致报警时，则输出点A反转，输出点B取输出点A的反逻辑
   IF xReady AND (NOT xManuAlmDisable) AND fbManuFall.Q THEN
	   xOutputA  := NOT xOutputA; 
	   xOutputB  := NOT xOutputA;
	   
	//手动操作生效时，判断输出点状态与自动命令是否一致，不一致时,置位手动操作执行中报警；一致时复位该报警。
	//当因安全条件不满足导致自动命令未执行时，可通过手动操作控制其动作执行,此时手动操作并不引起手动操作执行中报警。
   	   IF (stCylvar.xAutoCmd AND (NOT xManuAlmDisable) ) XOR xOutputB THEN
   	   	    f_xManuAlm  :=TRUE;
   	   ELSE 
   	   	    f_xManuAlm  :=FALSE;
   	   END_IF
   END_IF
   //2,手动操作时，如果满足安全条件且屏蔽了手自动不一致报警时，则自动控制点反转、复位手自动不一致报警，  
    IF xReady AND  xManuAlmDisable AND fbManuFall.Q THEN
   	    stCylvar.xAutoCmd  := NOT stCylvar.xAutoCmd ;
		f_xManuAlm  :=FALSE;		  	 	
    END_IF
   
   //自动命令置位时，如满足安全条件，则输出点A复位、 输出点B置位。
   IF xReady AND fbAutoRise.Q THEN
   	    xOutputA  :=FALSE;
		xOutputB  :=TRUE;
		
   END_IF
   //自动命令复位时，如满足安全条件，则输出点A置位、 输出点B复位。
   IF xReady AND fbAutoFall.Q THEN
   	    xOutputA  :=TRUE;
		xOutputB  :=FALSE;		
   END_IF
   
   
   //到位状态输出
   fbFrontTon(IN:=( NOT xOutputA ) AND xOutputB AND ( xFrontSensor OR xFrontSensorDisable ) AND ( NOT xBackSensor ) , PT:= WORD_TO_TIME ( wFrontDelay *10 ), Q=> stCylvar.xIsFront, ET=> );
   
   //原位状态输出
   fbBackTon(IN:= xOutputA  AND ( NOT xOutputB) AND ( NOT xFrontSensor ) AND ( xBackSensor OR xBackSensorDisable ) , PT:= WORD_TO_TIME ( wBackDelay *10 ) , Q=> stCylvar.xIsBack, ET=> );
   
   
   //报警复位
   fbResetRise(CLK:= xReset, Q=> );
   IF fbResetRise.Q THEN
   	   f_xNotRdyAlm := FALSE;
	   f_xFrontAlm := FALSE;
	   f_xBackAlm := FALSE;
	   f_xUncontrolledAlm := FALSE;
   
   END_IF
   
   
   //未满足安全条件报警
   //当手动操作或自动命令状态发生改变时，如果不能满足安全条件，则输出未满足安全条件报警
   IF ( fbManuFall.Q OR fbAutoRise.Q OR fbAutoFall.Q ) AND ( NOT xReady ) THEN
   	   f_xNotRdyAlm := TRUE; 
   END_IF
   
   
   //未在原位报警
   //自动命令变OFF后(上电后气缸处于自由状态时不判断)，延时5秒，如果原位标志未变为ON、且未发生手动操作和安全条件报警，则输出未到原位报警
   fbBackWait(IN:= ( NOT stCylvar.xAutoCmd ) AND ( xOutputA OR xOutputB ) , PT:= T#5S , Q=> , ET=> );
   fbBackFall(CLK:= stCylvar.xIsBack , Q=> );
   IF (( fbBackWait.Q AND (NOT stCylvar.xIsBack )) OR (( NOT stCylvar.xAutoCmd ) AND fbBackFall.Q )) AND  ( NOT f_xManuAlm ) AND  ( NOT f_xNotRdyAlm ) THEN
   	    f_xBackAlm := TRUE;
   END_IF
   
   
   //未在到位报警
   //自动命令变ON后，延时5秒，如果到位标志未变为ON、且未发生手动操作和安全条件报警，则输出未到位报警
   fbFrontWait(IN:= stCylvar.xAutoCmd , PT:= T#5S , Q=> , ET=> );
   fbFrontFall(CLK:= stCylvar.xIsFront, Q=> );
   IF ( ( fbFrontWait.Q AND ( NOT stCylvar.xIsFront ) ) OR (stCylvar.xAutoCmd AND fbFrontFall.Q )) AND ( NOT f_xManuAlm ) AND ( NOT f_xNotRdyAlm ) THEN
   	    f_xFrontAlm := TRUE;   
   END_IF      
   
   
   //不受控状态报警
   IF NOT ( xOutputA OR xOutputB ) THEN
   	    f_xUncontrolledAlm := TRUE;
   END_IF

END_FUNCTION_BLOCK

// Device/Application/FunctionBlock/FB_CylinderSingle
FUNCTION_BLOCK FB_CylinderSingle
VAR_IN_OUT
	stCylVar: CYLINDER_REF;
END_VAR
VAR_INPUT
	///安全条件
	xReady: BOOL;
	///报警复位
	xReset: BOOL;
	///手动控制,每on一次,则反转输出点状态
	xManuCmd: BOOL;
	///原位检测
	xBackSensor: BOOL;
	///到位检测
	xFrontSensor: BOOL;
	///手自动不一致报警无效
	xManuAlmDisable: BOOL;
	///原位检测无效
	xBackSensorDisable: BOOL;
	///到位检测无效
	xFrontSensorDisable: BOOL;
	///原位延时
	wBackDelay: WORD;
	///到位延时
	wFrontDelay: WORD;
END_VAR
VAR_OUTPUT
	xOutput: BOOL;
	///未满足安全条件报警
	f_xNotRdyAlm: BOOL;
	///手自动不一致报警	
	f_xManuAlm: BOOL;
	///未在原位报警
	f_xBackAlm: BOOL;
	///未到位报警
	f_xFrontAlm: BOOL;
END_VAR
VAR
	///获取自动控制的上升沿
	fbAutoRise: R_TRIG;
	///获取自动控制的下升沿
	fbAutoFall: F_TRIG;
	///获取手动控制的下升沿
	fbManuFall: F_TRIG;
	///获取复位信号的上升沿
	fbResetRise: R_TRIG;
	///原位状态延时,用于输出原位状态
	fbBackTon: TON;
	///到位状态延时,用于输出到位状态
	fbFrontTon: TON;
	///获取原位状态下降沿	
	fbBackFall: F_TRIG;
	///获取到位状态下降沿
	fbFrontFall: F_TRIG;
	///原位动作超时,用于输出未在原位位置报警
	fbBackWait: TON;
	///到位动作超时,用于输出未在到位位置报警
	fbFrontWait: TON;
END_VAR

   //初始化时复位输出点
   IF xReady AND stCylVar.xInit AND ( NOT f_xNotRdyAlm	) THEN
	    xOutput := FALSE;
	    f_xManuAlm  := FALSE;
	    stCylVar.xInit  := FALSE;
 
   END_IF


   //获取手动控制、自动控制的边沿信号
   fbManuFall(CLK:=xManuCmd , Q=> );
   fbAutoRise(CLK:=stCylvar.xAutoCmd , Q=> );
   fbAutoFall(CLK:=stCylvar.xAutoCmd , Q=> );
      
    //1,手动操作时，如果满足安全条件且未屏蔽了手自动不一致报警时，则输出点反转，  
    IF xReady AND (NOT xManuAlmDisable) AND fbManuFall.Q THEN
   	    xOutput  := NOT xOutput ;
		//手动操作生效时，判断输出点状态与自动命令是否一致，不一致时,置位手动操作执行中报警；一致时复位该报警。
	    //当因安全条件不满足导致自动命令未执行时，可通过手动操作控制其动作执行,此时手动操作并不引起手动操作执行中报警。
		 IF ( stCylvar.xAutoCmd ) XOR xOutput THEN
   	   	    f_xManuAlm  :=TRUE;
   	     ELSE 
   	   	    f_xManuAlm  :=FALSE;
   	     END_IF  	 	
     END_IF
	 
	//2,手动操作时，如果满足安全条件且屏蔽了手自动不一致报警时，则自动控制点反转、复位手自动不一致报警，  
    IF xReady AND  xManuAlmDisable AND fbManuFall.Q THEN
   	    stCylvar.xAutoCmd  := NOT stCylvar.xAutoCmd ;
		f_xManuAlm  :=FALSE;		  	 	
    END_IF
   
   
   
   //自动命令置位时，如果满足安全条件，则输出点置位
   IF xReady AND fbAutoRise.Q THEN
   	   xOutput  :=TRUE;
   END_IF
      
   //自动命令复位时，如满足安全条件，则输出点复位。
   IF xReady AND fbAutoFall.Q THEN
   	    xOutput  :=FALSE;		
   END_IF
   
   
   //原位状态输出
   fbBackTon(IN:= ( NOT xOutput) AND ( NOT xFrontSensor ) AND ( xBackSensor OR xBackSensorDisable ) , PT:= WORD_TO_TIME ( wBackDelay *10 ) , Q=> stCylvar.xIsBack, ET=> );
   
   
   //到位状态输出
   fbFrontTon(IN:= xOutput AND ( xFrontSensor OR xFrontSensorDisable ) AND ( NOT xBackSensor ) , PT:= WORD_TO_TIME ( wFrontDelay *10 ), Q=> stCylvar.xIsFront, ET=> );
      
	  
   //报警复位
   fbResetRise(CLK:= xReset, Q=> );
   IF fbResetRise.Q THEN
   	   f_xNotRdyAlm := FALSE;
	   f_xFrontAlm := FALSE;
	   f_xBackAlm := FALSE;
   
   END_IF
   
   
   //未满足安全条件报警
   //当手动操作或自动命令状态发生改变时，如果不能满足安全条件，则输出未满足安全条件报警
   IF ( fbManuFall.Q OR fbAutoRise.Q OR fbAutoFall.Q ) AND ( NOT xReady ) THEN
   	    f_xNotRdyAlm := TRUE; 
   END_IF
   
   
   //未在原位报警
   //自动命令变OFF后(上电后气缸处于自由状态时不判断)，延时5秒，如果原位标志未变为ON、且未发生手动操作和安全条件报警，则输出未到原位报警
   fbBackWait(IN:=  NOT stCylvar.xAutoCmd  , PT:= T#5S , Q=> , ET=> );
   fbBackFall(CLK:= stCylvar.xIsBack , Q=> );
   IF (( fbBackWait.Q AND (NOT stCylvar.xIsBack )) OR (( NOT stCylvar.xAutoCmd ) AND fbBackFall.Q )) AND  ( NOT f_xManuAlm ) AND  ( NOT f_xNotRdyAlm ) THEN
   	    f_xBackAlm := TRUE;
   END_IF
   
   
   //未到位报警
   //自动命令变ON后，延时5秒，如果到位标志未变为ON、且未发生手动操作和安全条件报警，则输出未到位报警
   fbFrontWait(IN:= stCylvar.xAutoCmd , PT:= T#5S , Q=> , ET=> );
   fbFrontFall(CLK:= stCylvar.xIsFront, Q=> );
   IF ( ( fbFrontWait.Q AND ( NOT stCylvar.xIsFront ) ) OR (stCylvar.xAutoCmd AND fbFrontFall.Q )) AND ( NOT f_xManuAlm ) AND ( NOT f_xNotRdyAlm ) THEN
   	    f_xFrontAlm := TRUE;   
   END_IF

END_FUNCTION_BLOCK
